FUNCTION_BLOCK PUBLIC LampStatusDecider
VAR_INPUT
	GivenTimer : TON;
	GivenTimer_1: TON;
	Giventimer_2: TON;
	
	CurrentStatus : BOOL;
END_VAR
VAR_OUTPUT
	NewStatus : BOOL;
END_VAR
VAR
END_VAR



	GivenTimer_1(IN:= NOT Giventimer_2.Q,PT:=T#500MS,Q=> );
	
	GivenTimer_2(IN:=GivenTimer_1.Q,PT:=T#500ms,Q=>);
	
	IF GivenTimer_1.Q THEN
	   NewStatus:=TRUE;	
	   ELSE
	   NewStatus:=FALSE;	   
	   END_IF
	
	




//IF GivenTimer.Q THEN
	//NewStatus := NOT CurrentStatus;
//END_IF

END_FUNCTION_BLOCK

(* stored: Version 1.1.0.1, ProductVersion 3.1.4022.16
   POU LampStatusDecider: Id {118a3368-d198-40a5-bb27-9fe0006960bd}, SpecialFunc None *)
